// TwinCAT 3 PLC project PanelSaw
// ProgramVersion: 3.1.4026.19
// libraries:
//   Tc2_Standard, * (Beckhoff Automation GmbH)
//   Tc2_System, * (Beckhoff Automation GmbH)
// project tree:
//   DUTs/ ST_MachineControl.TcDUT, ST_SawBladeData.TcDUT, ST_WoodPanelData.TcDUT
//   GVLs/ GVL_HMI.TcGVL, GVL_Parameters.TcGVL
//   / PlcTask.TcTTO
//   POUs/ FB_PressureBeam.TcPOU, FB_PusherClamp.TcPOU, FB_SafetyHandler.TcPOU, FB_SawCut.TcPOU, F_GetDefaultMainBlade.TcPOU, F_GetDefaultScoringBlade.TcPOU, MAIN.TcPOU, F_GetDefaultWoodPanel.TcPOU, PRG_INIT.TcPOU, PRG_MACHINE.TcPOU
// real-time tasks:
//   TASK PlcTask: cycle T#10ms, priority 20, ADS port 350
//   TASK PlcTask1: cycle T#10ms, priority 21, ADS port 351

CONFIGURATION PanelSaw
    RESOURCE PLC ON TwinCAT3
        TASK PlcTask(INTERVAL := T#10ms, PRIORITY := 21);
        PROGRAM MAIN WITH PlcTask : MAIN;
    END_RESOURCE
END_CONFIGURATION

// ---- DUTs/ST_MachineControl.TcDUT
TYPE ST_MachineControl :
STRUCT
	bPressureBeamLower : BOOL;
	bPressureBeamRaise : BOOL;
	bClamp : BOOL;
	bUnclamp: BOOL;
END_STRUCT
END_TYPE

// ---- DUTs/ST_SawBladeData.TcDUT
TYPE ST_SawBladeData :
STRUCT
	rBladeDiameter : REAL;
	rBladeRadius : REAL;
	rBladeThickness: REAL;
	sBladeType : STRING;
END_STRUCT
END_TYPE

// ---- DUTs/ST_WoodPanelData.TcDUT
TYPE ST_WoodPanelData :
STRUCT
	rPanelWidth : REAL; // Largura x <- 0 +>
	rPanelLength : REAL; // Comprimento y
	rPanelThickness: REAL ; // Espessura z
END_STRUCT
END_TYPE

// ---- GVLs/GVL_HMI.TcGVL
{attribute 'qualified_only'}
VAR_GLOBAL
	//SAW
	bMainSawActive : BOOL := FALSE;
	bScoringSawActive : BOOL := FALSE;
	rSawCarriagePosition : REAL;
	
	//CYCLE COMMAND
	bStartCycle : BOOL := FALSE;
	bStopCycle : BOOL := FALSE;
	
	nTotalCut : INT;
	nMachineState : INT;
	nCurrentCutIndex : INT;
	sStateDescription : STRING;
	arCutList : ARRAY[1..20] OF REAL;
	
	//TOOLS
	bPressureBeamActive : BOOL;     
	bPressureBeamLowered : BOOL;     
	bPressureBeamRaised : BOOL;    
	bPressureBeamMoving : BOOL;     
	bPressureBeamCommand : BOOL;
	
	bPusherClampActive : BOOL := FALSE;
	bPusherClampCommand : BOOL := FALSE;
	bPusherClampMoving : BOOL := FALSE;
	rPusherTargetPosition : REAL;
	rPusherFencePosition : REAL;
	
	bAirTablesActive : BOOL := FALSE;
	//SAFETY
	bSafetyFencesClosed : BOOL := FALSE;
	
	//EMERGENCY
	bEmergencyButton : BOOL := FALSE;
	bEmergencyResetButton : BOOL := FALSE;
END_VAR

// ---- GVLs/GVL_Parameters.TcGVL
{attribute 'qualified_only'}
VAR_GLOBAL
	stPanelData : ST_WoodPanelData;
	stMainBlade : ST_SawBladeData;
	stScoringBlade : ST_SawBladeData;
END_VAR

// ---- POUs/MAIN.TcPOU
PROGRAM MAIN
VAR
END_VAR

PRG_INIT();
PRG_MACHINE();

END_PROGRAM

// ---- POUs/PRG_INIT.TcPOU
PROGRAM PRG_INIT
VAR
	bProgramInit :BOOL := FALSE;
END_VAR

IF NOT bProgramInit THEN
	GVL_Parameters.stMainBlade := F_GetDefaultMainBlade();
	GVL_Parameters.stScoringBlade := F_GetDefaultScoringBlade();
	GVL_Parameters.stPanelData := F_GetDefaultWoodPanel();
	
	bProgramInit := TRUE;
END_IF

END_PROGRAM

// ---- POUs/F_GetDefaultMainBlade.TcPOU
FUNCTION F_GetDefaultMainBlade : ST_SawBladeData
VAR_INPUT
END_VAR
VAR
END_VAR

F_GetDefaultMainBlade.rBladeDiameter := 350.0;
F_GetDefaultMainBlade.rBladeRadius := F_GetDefaultMainBlade.rBladeDiameter / 2;
F_GetDefaultMainBlade.rBladeThickness := 3.2;
F_GetDefaultMainBlade.sBladeType := 'TCT Panel Saw Blade PI-521VS Premium';

END_FUNCTION

// ---- POUs/F_GetDefaultScoringBlade.TcPOU
FUNCTION F_GetDefaultScoringBlade : ST_SawBladeData
VAR_INPUT
END_VAR
VAR
END_VAR

F_GetDefaultScoringBlade.rBladeDiameter := 120.0;
F_GetDefaultScoringBlade.rBladeRadius := F_GetDefaultScoringBlade.rBladeDiameter / 2;
F_GetDefaultScoringBlade.rBladeThickness := 2.8;
F_GetDefaultScoringBlade.sBladeType := 'KWO split scoring saw blade';

END_FUNCTION

// ---- POUs/F_GetDefaultWoodPanel.TcPOU
FUNCTION F_GetDefaultWoodPanel : ST_WoodPanelData
VAR_INPUT
END_VAR
VAR
END_VAR

F_GetDefaultWoodPanel.rPanelWidth := 100.0; // Default width: 100mm
F_GetDefaultWoodPanel.rPanelLength := 500.0; // Default length: 500mm
F_GetDefaultWoodPanel.rPanelThickness := 5.0; // Default thickness: 5mm

END_FUNCTION

// ---- POUs/PRG_MACHINE.TcPOU
PROGRAM PRG_MACHINE
VAR	
	//Machine state
    nInternState : INT := 0;
    nSubState : INT := 0;
    nStateBeforeStop : INT := 0;
    
    // Function blocks
    fbPressureBeam : FB_PressureBeam;
    fbPusherClamp : FB_PusherClamp;
    fbSawCut : FB_SawCut; 
    fbSafety : FB_SafetyHandler;
    
    // Control structure
    stMachineControl : ST_MachineControl;
    
    // Cut tracking
    rCurrentCutPoint : REAL;
    nCurrentIndex : INT;
    
    // Safety timeout
    tonSafetyTimeout : TON;
END_VAR

fbSafety(
	bEmergencyButton := GVL_HMI.bEmergencyButton,
	bEmergencyResetButton := GVL_HMI.bEmergencyResetButton,
	bSafetyFencesClosed := GVL_HMI.bSafetyFencesClosed,
	nCurrentState :=nInternState
);
	IF fbSafety.bTriggerEmergency AND nInternState <>999 THEN
		nInternState := 999;
		SetSafeState();
		
	END_IF

IF GVL_HMI.bEmergencyResetButton THEN
    GVL_HMI.bEmergencyButton := FALSE;
    nInternState := 0;
    GVL_HMI.bEmergencyResetButton := FALSE;
END_IF
IF GVL_HMI.bStopCycle AND nInternState <> 4 THEN
    nStateBeforeStop := nInternState;
    nInternState := 4;
    SetSafeState();
END_IF

fbPressureBeam(
    bEnable := TRUE,
    bLowerCommand := stMachineControl.bPressureBeamLower OR GVL_HMI.bPressureBeamCommand,
    bRaiseCommand := stMachineControl.bPressureBeamRaise OR (NOT GVL_HMI.bPressureBeamCommand)
);

fbPusherClamp(
    bEnable := TRUE,
    bClampCommand := stMachineControl.bClamp OR GVL_HMI.bPusherClampCommand,
    bUnclampCommand := stMachineControl.bUnclamp OR (NOT GVL_HMI.bPusherClampCommand),
    rTargetPosition := GVL_HMI.rPusherTargetPosition,
    rCurrentPosition := GVL_HMI.rPusherFencePosition
);

GVL_HMI.bPressureBeamActive := fbPressureBeam.bActive;
GVL_HMI.bPressureBeamLowered := fbPressureBeam.bLowered;
GVL_HMI.bPressureBeamRaised := fbPressureBeam.bRaised;
GVL_HMI.bPressureBeamMoving := fbPressureBeam.bMoving;

GVL_HMI.bPusherClampActive := fbPusherClamp.bActive;
GVL_HMI.bPusherClampMoving := fbPusherClamp.bMoving;

GVL_HMI.nMachineState := nInternState;
GVL_HMI.nCurrentCutIndex := nCurrentIndex;
GVL_HMI.sStateDescription := fbSafety.sErrorMessage;

CASE nInternState OF
    0: StateIdle();
    1: StatePositioning();
    2: StateCutting();
    3: StateReturning();
    4: StateStopped();
    10: StateReleasing();
    999: StateEmergency();
END_CASE

ACTION SetSafeState:
stMachineControl.bPressureBeamRaise := TRUE;
stMachineControl.bPressureBeamLower := FALSE;
stMachineControl.bUnclamp := TRUE;
stMachineControl.bClamp := FALSE;
GVL_HMI.bScoringSawActive := FALSE;
GVL_HMI.bMainSawActive := FALSE;
fbSawCut(bExecute := FALSE, bResetTimer := TRUE);
END_ACTION

ACTION StateCutting:
GVL_HMI.sStateDescription := CONCAT('Cutting ', INT_TO_STRING(nCurrentIndex));

stMachineControl.bPressureBeamLower := TRUE;
stMachineControl.bPressureBeamRaise := FALSE;
stMachineControl.bClamp := TRUE;
stMachineControl.bUnclamp := FALSE;

fbSawCut(
    bExecute := TRUE,
    rPanelWidth := GVL_Parameters.stPanelData.rPanelWidth,
    bResetTimer := FALSE
);

IF fbSawCut.bBusy THEN
    GVL_HMI.bScoringSawActive := TRUE;
    GVL_HMI.bMainSawActive := TRUE;
END_IF

IF fbSawCut.bError THEN
    GVL_HMI.sStateDescription := 'Error during cutting operation';
    SetSafeState();
    nInternState := 999;
    nSubState := 0;
ELSIF fbSawCut.bDone THEN
    GVL_HMI.bScoringSawActive := FALSE;
    GVL_HMI.bMainSawActive := FALSE;
    fbSawCut(bExecute := FALSE);
    nInternState := 10;
    nSubState := 0;
END_IF
END_ACTION

ACTION StateEmergency:
GVL_HMI.nMachineState := nInternState;
GVL_HMI.nCurrentCutIndex := nCurrentIndex;

IF nInternState = 999 THEN
    GVL_HMI.sStateDescription := fbSafety.sErrorMessage;
END_IF
END_ACTION

ACTION StateIdle:
GVL_HMI.sStateDescription := 'Machine Idling.';
SetSafeState();

nCurrentIndex := 0;
nSubState := 0;

IF GVL_HMI.bStartCycle THEN
    GVL_HMI.bStartCycle := FALSE;
    IF GVL_HMI.nTotalCut > 0 AND GVL_HMI.nTotalCut <= 20 THEN
        IF fbSafety.bAllowOperation THEN
            nCurrentIndex := 1;
            nInternState := 1;
        ELSE
            GVL_HMI.sStateDescription := 'ERROR: Safety conditions not met.';
        END_IF
    END_IF
END_IF
END_ACTION

ACTION StatePositioning:
IF GVL_HMI.nTotalCut < 1 OR GVL_HMI.nTotalCut > 20 THEN
    GVL_HMI.sStateDescription := 'ERROR: Cut Index out of range';
    nInternState := 999;
    RETURN;
END_IF

rCurrentCutPoint := GVL_HMI.arCutList[nCurrentIndex] + GVL_Parameters.stMainBlade.rBladeThickness / 2;
GVL_HMI.rPusherTargetPosition := rCurrentCutPoint;

tonSafetyTimeout(IN := TRUE, PT := T#60S);
IF tonSafetyTimeout.Q THEN
    GVL_HMI.sStateDescription := 'ERROR: Positioning timeout';
    nInternState := 999;
    tonSafetyTimeout(IN := FALSE);
    RETURN;
END_IF

CASE nSubState OF
    0:
        GVL_HMI.sStateDescription := CONCAT('Positioning for cut ', INT_TO_STRING(nCurrentIndex));
        
        stMachineControl.bPressureBeamRaise := TRUE;
        stMachineControl.bPressureBeamLower := FALSE;
        stMachineControl.bUnclamp := TRUE;
        stMachineControl.bClamp := FALSE;
        
        IF ABS(GVL_HMI.rPusherFencePosition - rCurrentCutPoint) > 0.1 THEN
            IF GVL_HMI.rPusherFencePosition < rCurrentCutPoint THEN
                GVL_HMI.rPusherFencePosition := GVL_HMI.rPusherFencePosition + 0.1;
            ELSE
                GVL_HMI.rPusherFencePosition := GVL_HMI.rPusherFencePosition - 0.1;
            END_IF
        ELSE
            nSubState := 1;
        END_IF
        
    1:
        GVL_HMI.sStateDescription := 'Lowering pressure beam...';
        stMachineControl.bPressureBeamLower := TRUE;
        stMachineControl.bPressureBeamRaise := FALSE;
        
        IF fbPressureBeam.bLowered THEN
            nSubState := 2;
        END_IF
        
    2:
        GVL_HMI.sStateDescription := 'Activating clamp...';
        stMachineControl.bClamp := TRUE;
        stMachineControl.bUnclamp := FALSE;
        
        IF fbPusherClamp.bActive THEN
            tonSafetyTimeout(IN := FALSE);
            nInternState := 2;
            nSubState := 0;
        END_IF
END_CASE
END_ACTION

ACTION StateReleasing:
CASE nSubState OF
    0: // Raise beam
        GVL_HMI.sStateDescription := 'Raising pressure beam...';
        stMachineControl.bPressureBeamRaise := TRUE;
        stMachineControl.bPressureBeamLower := FALSE;
        stMachineControl.bClamp := TRUE;
        
        IF fbPressureBeam.bRaised THEN
            nSubState := 1;
        END_IF
        
    1: // Unclamp
        GVL_HMI.sStateDescription := 'Releasing clamp...';
        stMachineControl.bUnclamp := TRUE;
        stMachineControl.bClamp := FALSE;
        
        IF fbPusherClamp.bUnclamped THEN
            nCurrentIndex := nCurrentIndex + 1;
            
            IF nCurrentIndex > GVL_HMI.nTotalCut THEN
                nInternState := 3;
            ELSE
                nInternState := 1;
            END_IF
            nSubState := 0;
        END_IF
END_CASE
END_ACTION

ACTION StateReturning:
GVL_HMI.sStateDescription := 'Returning to home position...';
SetSafeState();

IF GVL_HMI.rPusherFencePosition > 0.0 THEN
    GVL_HMI.rPusherFencePosition := GVL_HMI.rPusherFencePosition - 0.1;
ELSE
    GVL_HMI.rPusherFencePosition := 0.0;
    GVL_HMI.sStateDescription := 'Cycle complete!';
    nInternState := 0;
END_IF
END_ACTION

ACTION StateStopped:
GVL_HMI.sStateDescription := 'Machine stopped.';
SetSafeState();

IF NOT GVL_HMI.bStopCycle THEN
    nInternState := nStateBeforeStop;
END_IF
END_ACTION

END_PROGRAM

// ---- POUs/FB_PressureBeam.TcPOU
FUNCTION_BLOCK FB_PressureBeam
VAR_INPUT
	bEnable : BOOL;
	bLowerCommand : BOOL;
	bRaiseCommand : BOOL;
	tLowerTime : TIME := T#2S;
	tRaiseTime : TIME := T#1S500MS;
END_VAR
VAR_OUTPUT
	bLowered: BOOL;
	bRaised : BOOL;
	bMoving : BOOL;
	bError : BOOL;
	bActive : BOOL;
END_VAR
VAR
	eState : (IDLE, LOWERING, LOWERED, RAISING, ERROR) := IDLE;
	tonLower : TON;
	tonRaise : TON;
	tonTimeout : TON;
END_VAR

CASE eState OF
	IDLE:
		bMoving := FALSE;
		bLowered := FALSE;
		bRaised := TRUE;
		bActive := FALSE;
		tonLower(IN := FALSE);
		tonRaise(IN := FALSE);
		
		IF bEnable AND bLowerCommand THEN
			eSTATE := LOWERING;
		END_IF
	LOWERING:
		bMoving := TRUE;
		bRaised := FALSE;
		tonLower(IN := TRUE, PT := tLowerTime);
		
		IF tonLower.Q THEN
			eState := LOWERED;
			tonLower(IN := FALSE);
		END_IF
	LOWERED:
		bMoving := FALSE;
		bLowered := TRUE;
		bActive := TRUE;
		IF bRaiseCommand OR NOT bEnable THEN
			eState := RAISING;
		END_IF
	RAISING:
		bMoving := TRUE;
		bLowered := FALSE;
		tonRaise(IN := TRUE, PT := tRaiseTime);
		
		IF tonRaise.Q THEN
			eState := IDLE;
			tonRaise(IN := FALSE);
		END_IF
	ERROR:
		bError := TRUE;
		bMoving := FALSE;
		
		IF NOT bEnable THEN
			eState := IDLE;
			bError := FALSE;
		END_IF		
END_CASE

END_FUNCTION_BLOCK

// ---- POUs/FB_PusherClamp.TcPOU
FUNCTION_BLOCK FB_PusherClamp
VAR_INPUT
	bEnable : BOOL;
	bClampCommand : BOOL;
	bUnclampCommand : BOOL;
	rTargetPosition : REAL;
	rCurrentPosition : REAL;
	rTolerance : REAL := 0.2;
	tClampTime : TIME := T#1S;
	tUnclampTime : TIME := T#800MS;
END_VAR
VAR_OUTPUT
	bUnclamped : BOOL;
	bAtPosition : BOOL;
	bMoving : BOOL;
	bError : BOOL;
	bActive : BOOL;
END_VAR
VAR
	eState : (IDLE, POSITIONING, CLAMPING, CLAMPED, UNCLAMPING, ERROR) := IDLE;
	tonClamp : TON;
	tonUnclamp : TON;
	tonPositionTimeout : TON;
END_VAR

bAtPosition := ABS(rCurrentPosition - rTargetPosition) <= rTolerance;

CASE eState OF
    IDLE:
        bMoving := FALSE;
        bUnclamped := TRUE;
        bActive := FALSE;
        tonClamp(IN := FALSE);
        tonUnclamp(IN := FALSE);
        
        IF bEnable AND bClampCommand AND bAtPosition THEN
            eState := CLAMPING;
        END_IF
        
    CLAMPING:
        bMoving := FALSE;
        tonClamp(IN := TRUE, PT := tClampTime);
        
        IF tonClamp.Q THEN
            eState := CLAMPED;
            tonClamp(IN := FALSE);
        END_IF
        
    CLAMPED:
        bActive := TRUE;
        bMoving := FALSE;
        
        IF bUnclampCommand OR NOT bEnable THEN
            eState := UNCLAMPING;
        END_IF
        
    UNCLAMPING:
		bUnclamped := FALSE;
		bActive := FALSE;
        tonUnclamp(IN := TRUE, PT := tUnclampTime);
        
        IF tonUnclamp.Q THEN
			bUnclamped := TRUE;
            eState := IDLE;
            tonUnclamp(IN := FALSE);
        END_IF
        
    ERROR:
        bError := TRUE;
        bMoving := FALSE;
        IF NOT bEnable THEN
            eState := IDLE;
            bError := FALSE;
        END_IF
END_CASE

END_FUNCTION_BLOCK

// ---- POUs/FB_SawCut.TcPOU
FUNCTION_BLOCK FB_SawCut
VAR_INPUT
    bExecute : BOOL;          // Start cut operation
    rPanelWidth : LREAL;      // Panel width in mm
    bResetTimer : BOOL;       // Reset timer
END_VAR

VAR_OUTPUT
    bDone : BOOL;             // Cut complete
    bBusy : BOOL;             // Cut in progress
    bError : BOOL;            // Error occurred
    tRemainingTime : TIME;    // Time remaining
END_VAR

VAR
    tonCutTimer : TON;                  // Timer that counts cut duration
    tCalculatedCutTime : TIME;          // How long this cut should take
    rCutTimePerMM : LREAL := 0.05;      // 50ms per mm (adjust for your machine speed)
    tMinCutTime : TIME := T#2S;         // Never cut less than 2 seconds
    tMaxCutTime : TIME := T#30S;        // Never cut more than 30 seconds
    bExecuteOld : BOOL := FALSE;        // Previous value of bExecute
    nState : INT := 0;                  // 0=IDLE, 10=CUTTING, 20=DONE
END_VAR

CASE nState OF
    0: // IDLE
        bDone := FALSE;
        bBusy := FALSE;
        
        IF bExecute AND NOT bExecuteOld THEN
            tCalculatedCutTime := LREAL_TO_TIME(rPanelWidth * rCutTimePerMM * 1000.0);
            IF tCalculatedCutTime < tMinCutTime THEN
                tCalculatedCutTime := tMinCutTime;
            ELSIF tCalculatedCutTime > tMaxCutTime THEN
                tCalculatedCutTime := tMaxCutTime;
            END_IF
            
            nState := 10;
        END_IF
        
    10: // CUTTING
        bBusy := TRUE;
        tonCutTimer(IN := TRUE, PT := tCalculatedCutTime);
        tRemainingTime := tCalculatedCutTime - tonCutTimer.ET;
        
        IF tonCutTimer.Q THEN
			tonCutTimer(IN := FALSE);
            nState := 20;
        END_IF
        
        IF NOT bExecute OR bResetTimer THEN
			tonCutTimer(IN := FALSE);
            nState := 0;
        END_IF
        
    20: // DONE
        bDone := TRUE;
        bBusy := FALSE;
        tonCutTimer(IN := FALSE);
        
        IF NOT bExecute THEN
            nState := 0;
        END_IF
        
END_CASE
bExecuteOld := bExecute;

END_FUNCTION_BLOCK

// ---- POUs/FB_SafetyHandler.TcPOU
FUNCTION_BLOCK FB_SafetyHandler
VAR_INPUT
	bEmergencyButton : BOOL;
	bEmergencyResetButton : BOOL;
	bSafetyFencesClosed : BOOL;
	nCurrentState : INT;
END_VAR
VAR_OUTPUT
	bTriggerEmergency : BOOL;
	bAllowOperation : BOOL;
	sErrorMessage : STRING;
END_VAR
VAR
END_VAR

bAllowOperation := bSafetyFencesClosed AND NOT bEmergencyButton;
bTriggerEmergency := bEmergencyButton OR (NOT bSafetyFencesClosed AND(nCurrentState = 1 OR nCurrentState = 2));

IF bEmergencyButton THEN
	sErrorMessage := '***EMERGENCY STOP***';
ELSIF NOT bSafetyFencesClosed THEN
	sErrorMessage := 'EMERGENCY: Safety fence opened during operation!';
END_IF

END_FUNCTION_BLOCK
